FUNCTION_BLOCK PressureGradient
VAR_INPUT
	TotalVolume: LREAL;
	BulkModulus: LREAL;
	FlowrateIn: LREAL;
	FlowrateOut: LREAL;
END_VAR
VAR_OUTPUT
	PressureGradientb : LREAL;
	PressureGradientPascal : LREAL;
END_VAR
VAR
END_VAR


(* Outputs for Atomic SubSystem: '<Root>/PressureGradient' *)
(* Outport: '<Root>/PressureGradientb' incorporates:
 *  Gain: '<S1>/Conv.2'
 *  Product: '<S1>/Product'
 *  Product: '<S1>/Product1'
 *  Sum: '<S1>/Sum' *)
PressureGradientb := ((FlowrateIn - FlowrateOut) * 1.6666666666666667E-5) * (BulkModulus / TotalVolume);
(* End of Outputs for SubSystem: '<Root>/PressureGradient' *)
//Gives PressureGradient in [Bar/s]

PressureGradientPascal := PressureGradientb*1E5;      //Multiplies to get Pascal

END_FUNCTION_BLOCK

(* stored: Version 1.1.0.1, ProductVersion 3.1.4024.9
   POU PressureGradient: Id {0ae25e94-6017-429e-9462-38875999b492}, SpecialFunc None *)
